FUNCTION_BLOCK InnerCompositeBlock
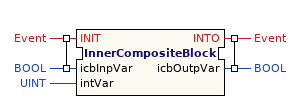
  EVENT_INPUT
    INIT WITH icbInpVar;
  END_EVENT
  EVENT_OUTPUT
    INTO WITH icbOutpVar;
  END_EVENT
  VAR_INPUT
    icbInpVar : BOOL;
    intVar : UINT;
  END_VAR
  VAR_OUTPUT
    icbOutpVar : BOOL;
  END_VAR
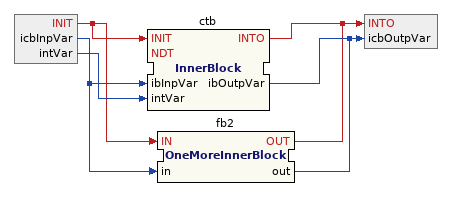
  FBS
    ctb : InnerBlock;
    fb2 : OneMoreInnerBlock;
  END_FBS
  EVENT_CONNECTIONS
    INIT TO ctb.INIT;
    ctb.INTO TO INTO;
    INIT TO fb2.IN;
    fb2.OUT TO INTO;
  END_CONNECTIONS
  DATA_CONNECTIONS
    icbInpVar TO ctb.ibInpVar;
    ctb.ibOutpVar TO icbOutpVar;
    icbInpVar TO fb2.in;
    fb2.out TO icbOutpVar;
    intVar TO ctb.intVar;
  END_CONNECTIONS
END_FUNCTION_BLOCK
